// TwinCAT 3 PLC project Komplett
// ProgramVersion: 3.1.4022.1
// libraries:
//   Tc2_Standard, * (Beckhoff Automation GmbH)
//   Tc2_System, * (Beckhoff Automation GmbH)
//   Tc3_Module, * (Beckhoff Automation GmbH)
// project tree:
//   GVLs/ AN.TcGVL, DIO.TcGVL, dSub.TcGVL
//   / PlcTask.TcTTO (not stored)
//   POUs/ DoppelLauflicht.TcPOU, Komplett.TcPOU, Lauflicht.TcPOU, MAIN.TcPOU
// real-time tasks:
//   TASK PlcTask: cycle T#10ms, priority 20, ADS port 350
// motion (NC):
//   TASK NC-Task 1 SAF: cycle T#2ms, priority 4, ADS port 501
//   TASK NC-Task 1 SVB: cycle T#10ms, priority 8, ADS port 511
//   AXIS Axis 1 (id 1)
//     OtherSettings: AllowMotionCmdToSlave=true
//     encoder EncType=4
//       EncPara: MaxCount=#x0000ffff
//         Inc: RefSoftSyncMask=#x0000ffff
//     drive DrvType=24
//       Analog: ScaleFactorActTorque=0.1
//       TimeComp: TaskDelayCycles=1
//     controller CtrType=1
//       CtrPara: PriorControlFactor=1
//         Observer: BandWidth=20
//   AXIS Axis 2 (id 2)
//     OtherSettings: AllowMotionCmdToSlave=true
//     encoder EncType=4
//       EncPara: MaxCount=#x0000ffff
//         Inc: RefSoftSyncMask=#x0000ffff
//     drive DrvType=24
//       Analog: ScaleFactorActTorque=0.1
//       TimeComp: TaskDelayCycles=1
//     controller CtrType=1
//       CtrPara: PriorControlFactor=1
//         Observer: BandWidth=20
//   AXIS Axis 3 (id 3)
//     OtherSettings: AllowMotionCmdToSlave=true
//     encoder EncType=4
//       EncPara: MaxCount=#x0000ffff
//     drive DrvType=23
//       Analog: ScaleFactorActTorque=0.1
//       TimeComp: TaskDelayCycles=1
//     controller CtrType=1
//       CtrPara: PriorControlFactor=1
//         Observer: BandWidth=20
//   AXIS Axis 4 (id 4)
//     OtherSettings: AllowMotionCmdToSlave=true
//     encoder EncType=4
//       EncPara: MaxCount=#x0000ffff
//     drive DrvType=23
//       Analog: ScaleFactorActTorque=0.1
//       TimeComp: TaskDelayCycles=1
//     controller CtrType=1
//       CtrPara: PriorControlFactor=1
//         Observer: BandWidth=20
//   AXIS Axis 5 (id 5)
//     OtherSettings: AllowMotionCmdToSlave=true
//     encoder EncType=19
//       EncPara: MaxCount=#xffffffff
//     drive DrvType=16
//       DrvPara: MaxCount=#xffffffff
//         Analog: ScaleFactorActTorque=0.1
//         TimeComp: TaskDelayCycles=1
//     controller CtrType=1
//       CtrPara: PriorControlFactor=1
//         Observer: BandWidth=20
//   AXIS Axis 6 (id 6)
//     OtherSettings: AllowMotionCmdToSlave=true
//     encoder EncType=19
//       EncPara: MaxCount=#xffffffff
//     drive DrvType=16
//       DrvPara: MaxCount=#xffffffff
//         Analog: ScaleFactorActTorque=0.1
//         TimeComp: TaskDelayCycles=1
//     controller CtrType=1
//       CtrPara: PriorControlFactor=1
//         Observer: BandWidth=20
// I/O:
//   DEVICE Device 1 (EtherCAT), AmsNetId 5.35.139.20.2.1
//     Term 1 (EK1200) [EK1200-5000 EtherCAT Power supply (2A E-Bus)]
//       Term 2 (EL1809) [EL1809 16Ch. Dig. Input 24V, 3ms]
//       Term 3 (EL1809) [EL1809 16Ch. Dig. Input 24V, 3ms]
//       Term 4 (EL2809) [EL2809 16Ch. Dig. Output 24V, 0.5A]
//       Term 5 (EL2809) [EL2809 16Ch. Dig. Output 24V, 0.5A]
//       Term 6 (EL3064) [EL3064 4Ch. Ana. Input 0-10V]
//       Term 7 (EL4034) [EL4034 4Ch. Ana. Output +/-10V, 12bit]
//       Term 8 (EL7031) [EL7031 1Ch. Stepper motor output stage (24V, 1.5A)]
//       Term 9 (EL7031) [EL7031 1Ch. Stepper motor output stage (24V, 1.5A)]
//       Term 10 (EL7332) [EL7332 2Ch. DC motor output stage (24V, 1.5A)]
//       Term 11 (EL7201-0010) [EL7201-0010 1Ch. MDP742 Servo motor output stage with OCT (50V, 4A)]
//       Term 12 (EL7201-0010) [EL7201-0010 1Ch. MDP742 Servo motor output stage with OCT (50V, 4A)]
//       Term 26 (EL6090) [EL6090 Display terminal]
//       Term 27 (EK1110) [EK1110 EtherCAT extension]
// variable links:
//   NC-Task 1 SAF/Axes/Axis 1 <-> Device 1 (EtherCAT)/Term 1 (EK1200)/Term 8 (EL7031)
//     Drive/Inputs/In/nState1 @bit 3 <-> STM Status/Status/Error
//     Drive/Inputs/In/nState1 @bit 5 <-> STM Status/Status/Moving negative
//     Drive/Inputs/In/nState1 @bit 4 <-> STM Status/Status/Moving positive
//     Drive/Inputs/In/nState1 @bit 1 <-> STM Status/Status/Ready
//     Drive/Inputs/In/nState1 <-> STM Status/Status/Ready to enable
//     Drive/Inputs/In/nState1 @bit 6 <-> STM Status/Status/Torque reduced
//     Drive/Inputs/In/nState1 @bit 2 <-> STM Status/Status/Warning
//     Drive/Inputs/In/nState2 @bit 3 <-> STM Status/Status/Digital input 1
//     Drive/Inputs/In/nState2 @bit 4 <-> STM Status/Status/Digital input 2
//     Drive/Inputs/In/nState2 @bit 5 <-> STM Status/Status/Sync error
//     Drive/Inputs/In/nState2 @bit 7 <-> STM Status/Status/TxPDO Toggle
//     Drive/Inputs/In/nState4 @bit 1 <-> WcState/InputToggle
//     Drive/Inputs/In/nState4 <-> WcState/WcState
//     Drive/Outputs/Out/nCtrl1 <-> STM Control/Control/Enable
//     Drive/Outputs/Out/nCtrl1 @bit 2 <-> STM Control/Control/Reduce torque
//     Drive/Outputs/Out/nCtrl1 @bit 1 <-> STM Control/Control/Reset
//     Drive/Outputs/Out/nDataOut2[0] <-> STM Velocity/Velocity
//     Enc/Inputs/In/nDataIn1[0] <-> ENC Status compact/Counter value
//     Enc/Inputs/In/nDataIn2[0] <-> ENC Status compact/Latch value
//     Enc/Inputs/In/nState1 @bit 4 <-> ENC Status compact/Status/Counter overflow
//     Enc/Inputs/In/nState1 @bit 3 <-> ENC Status compact/Status/Counter underflow
//     Enc/Inputs/In/nState1 @bit 1 <-> ENC Status compact/Status/Latch extern valid
//     Enc/Inputs/In/nState1 @bit 2 <-> ENC Status compact/Status/Set counter done
//     Enc/Inputs/In/nState2 @bit 4 <-> ENC Status compact/Status/Status of extern latch
//     Enc/Inputs/In/nState2 @bit 5 <-> ENC Status compact/Status/Sync error
//     Enc/Inputs/In/nState2 @bit 7 <-> ENC Status compact/Status/TxPDO Toggle
//     Enc/Inputs/In/nState4 @bit 1 <-> WcState/InputToggle
//     Enc/Inputs/In/nState4 <-> WcState/WcState
//     Enc/Outputs/Out/nCtrl1 @bit 3 <-> ENC Control compact/Control/Enable latch extern on negative edge
//     Enc/Outputs/Out/nCtrl1 @bit 1 <-> ENC Control compact/Control/Enable latch extern on positive edge
//     Enc/Outputs/Out/nCtrl1 @bit 2 <-> ENC Control compact/Control/Set counter
//     Enc/Outputs/Out/nDataOut1[0] <-> ENC Control compact/Set counter value
//   NC-Task 1 SAF/Axes/Axis 2 <-> Device 1 (EtherCAT)/Term 1 (EK1200)/Term 9 (EL7031)
//     Drive/Inputs/In/nState1 @bit 3 <-> STM Status/Status/Error
//     Drive/Inputs/In/nState1 @bit 5 <-> STM Status/Status/Moving negative
//     Drive/Inputs/In/nState1 @bit 4 <-> STM Status/Status/Moving positive
//     Drive/Inputs/In/nState1 @bit 1 <-> STM Status/Status/Ready
//     Drive/Inputs/In/nState1 <-> STM Status/Status/Ready to enable
//     Drive/Inputs/In/nState1 @bit 6 <-> STM Status/Status/Torque reduced
//     Drive/Inputs/In/nState1 @bit 2 <-> STM Status/Status/Warning
//     Drive/Inputs/In/nState2 @bit 3 <-> STM Status/Status/Digital input 1
//     Drive/Inputs/In/nState2 @bit 4 <-> STM Status/Status/Digital input 2
//     Drive/Inputs/In/nState2 @bit 5 <-> STM Status/Status/Sync error
//     Drive/Inputs/In/nState2 @bit 7 <-> STM Status/Status/TxPDO Toggle
//     Drive/Inputs/In/nState4 @bit 1 <-> WcState/InputToggle
//     Drive/Inputs/In/nState4 <-> WcState/WcState
//     Drive/Outputs/Out/nCtrl1 <-> STM Control/Control/Enable
//     Drive/Outputs/Out/nCtrl1 @bit 2 <-> STM Control/Control/Reduce torque
//     Drive/Outputs/Out/nCtrl1 @bit 1 <-> STM Control/Control/Reset
//     Drive/Outputs/Out/nDataOut2[0] <-> STM Velocity/Velocity
//     Enc/Inputs/In/nDataIn1[0] <-> ENC Status compact/Counter value
//     Enc/Inputs/In/nDataIn2[0] <-> ENC Status compact/Latch value
//     Enc/Inputs/In/nState1 @bit 4 <-> ENC Status compact/Status/Counter overflow
//     Enc/Inputs/In/nState1 @bit 3 <-> ENC Status compact/Status/Counter underflow
//     Enc/Inputs/In/nState1 @bit 1 <-> ENC Status compact/Status/Latch extern valid
//     Enc/Inputs/In/nState1 @bit 2 <-> ENC Status compact/Status/Set counter done
//     Enc/Inputs/In/nState2 @bit 4 <-> ENC Status compact/Status/Status of extern latch
//     Enc/Inputs/In/nState2 @bit 5 <-> ENC Status compact/Status/Sync error
//     Enc/Inputs/In/nState2 @bit 7 <-> ENC Status compact/Status/TxPDO Toggle
//     Enc/Inputs/In/nState4 @bit 1 <-> WcState/InputToggle
//     Enc/Inputs/In/nState4 <-> WcState/WcState
//     Enc/Outputs/Out/nCtrl1 @bit 3 <-> ENC Control compact/Control/Enable latch extern on negative edge
//     Enc/Outputs/Out/nCtrl1 @bit 1 <-> ENC Control compact/Control/Enable latch extern on positive edge
//     Enc/Outputs/Out/nCtrl1 @bit 2 <-> ENC Control compact/Control/Set counter
//     Enc/Outputs/Out/nDataOut1[0] <-> ENC Control compact/Set counter value
//   NC-Task 1 SAF/Axes/Axis 3 <-> Device 1 (EtherCAT)/Term 1 (EK1200)/Term 10 (EL7332)
//     Drive/Inputs/In/nState1 @bit 3 <-> DCM Status Channel 1/Status/Error
//     Drive/Inputs/In/nState1 @bit 5 <-> DCM Status Channel 1/Status/Moving negative
//     Drive/Inputs/In/nState1 @bit 4 <-> DCM Status Channel 1/Status/Moving positive
//     Drive/Inputs/In/nState1 @bit 1 <-> DCM Status Channel 1/Status/Ready
//     Drive/Inputs/In/nState1 <-> DCM Status Channel 1/Status/Ready to enable
//     Drive/Inputs/In/nState1 @bit 6 <-> DCM Status Channel 1/Status/Torque reduced
//     Drive/Inputs/In/nState1 @bit 2 <-> DCM Status Channel 1/Status/Warning
//     Drive/Inputs/In/nState2 @bit 3 <-> DCM Status Channel 1/Status/Digital input 1
//     Drive/Inputs/In/nState2 @bit 4 <-> DCM Status Channel 1/Status/Digital input 2
//     Drive/Inputs/In/nState2 @bit 5 <-> DCM Status Channel 1/Status/Sync error
//     Drive/Inputs/In/nState2 @bit 7 <-> DCM Status Channel 1/Status/TxPDO Toggle
//     Drive/Inputs/In/nState4 @bit 1 <-> WcState/InputToggle
//     Drive/Inputs/In/nState4 <-> WcState/WcState
//     Drive/Outputs/Out/nCtrl1 <-> DCM Control Channel 1/Control/Enable
//     Drive/Outputs/Out/nCtrl1 @bit 2 <-> DCM Control Channel 1/Control/Reduce torque
//     Drive/Outputs/Out/nCtrl1 @bit 1 <-> DCM Control Channel 1/Control/Reset
//     Drive/Outputs/Out/nDataOut2[0] <-> DCM Velocity Channel 1/Velocity
//   NC-Task 1 SAF/Axes/Axis 4 <-> Device 1 (EtherCAT)/Term 1 (EK1200)/Term 10 (EL7332)
//     Drive/Inputs/In/nState1 @bit 3 <-> DCM Status Channel 2/Status/Error
//     Drive/Inputs/In/nState1 @bit 5 <-> DCM Status Channel 2/Status/Moving negative
//     Drive/Inputs/In/nState1 @bit 4 <-> DCM Status Channel 2/Status/Moving positive
//     Drive/Inputs/In/nState1 @bit 1 <-> DCM Status Channel 2/Status/Ready
//     Drive/Inputs/In/nState1 <-> DCM Status Channel 2/Status/Ready to enable
//     Drive/Inputs/In/nState1 @bit 6 <-> DCM Status Channel 2/Status/Torque reduced
//     Drive/Inputs/In/nState1 @bit 2 <-> DCM Status Channel 2/Status/Warning
//     Drive/Inputs/In/nState2 @bit 3 <-> DCM Status Channel 2/Status/Digital input 1
//     Drive/Inputs/In/nState2 @bit 4 <-> DCM Status Channel 2/Status/Digital input 2
//     Drive/Inputs/In/nState2 @bit 5 <-> DCM Status Channel 2/Status/Sync error
//     Drive/Inputs/In/nState2 @bit 7 <-> DCM Status Channel 2/Status/TxPDO Toggle
//     Drive/Inputs/In/nState4 @bit 1 <-> WcState/InputToggle
//     Drive/Inputs/In/nState4 <-> WcState/WcState
//     Drive/Outputs/Out/nCtrl1 <-> DCM Control Channel 2/Control/Enable
//     Drive/Outputs/Out/nCtrl1 @bit 2 <-> DCM Control Channel 2/Control/Reduce torque
//     Drive/Outputs/Out/nCtrl1 @bit 1 <-> DCM Control Channel 2/Control/Reset
//     Drive/Outputs/Out/nDataOut2[0] <-> DCM Velocity Channel 2/Velocity
//   NC-Task 1 SAF/Axes/Axis 5 <-> Device 1 (EtherCAT)/Term 1 (EK1200)/Term 11 (EL7201-0010)
//     Drive/Inputs/In/nDcOutputTime <-> InfoData/DcOutputShift
//     Drive/Inputs/In/nState1 <-> DRV Statusword/Statusword
//     Drive/Inputs/In/nState2 <-> DRV Statusword/Statusword @bit 8
//     Drive/Inputs/In/nState4 @bit 1 <-> WcState/InputToggle
//     Drive/Inputs/In/nState4 <-> WcState/WcState
//     Drive/Outputs/Out/nCtrl1 <-> DRV Controlword/Controlword
//     Drive/Outputs/Out/nCtrl2 <-> DRV Controlword/Controlword @bit 8
//     Drive/Outputs/Out/nDataOut2 <-> DRV Target velocity/Target velocity
//     Enc/Inputs/In/nDataIn1 <-> FB Position/Position
//     Enc/Inputs/In/nDcInputTime <-> InfoData/DcInputShift
//     Enc/Inputs/In/nState4 @bit 1 <-> WcState/InputToggle
//     Enc/Inputs/In/nState4 <-> WcState/WcState
//   NC-Task 1 SAF/Axes/Axis 6 <-> Device 1 (EtherCAT)/Term 1 (EK1200)/Term 12 (EL7201-0010)
//     Drive/Inputs/In/nDcOutputTime <-> InfoData/DcOutputShift
//     Drive/Inputs/In/nState1 <-> DRV Statusword/Statusword
//     Drive/Inputs/In/nState2 <-> DRV Statusword/Statusword @bit 8
//     Drive/Inputs/In/nState4 @bit 1 <-> WcState/InputToggle
//     Drive/Inputs/In/nState4 <-> WcState/WcState
//     Drive/Outputs/Out/nCtrl1 <-> DRV Controlword/Controlword
//     Drive/Outputs/Out/nCtrl2 <-> DRV Controlword/Controlword @bit 8
//     Drive/Outputs/Out/nDataOut2 <-> DRV Target velocity/Target velocity
//     Enc/Inputs/In/nDataIn1 <-> FB Position/Position
//     Enc/Inputs/In/nDcInputTime <-> InfoData/DcInputShift
//     Enc/Inputs/In/nState4 @bit 1 <-> WcState/InputToggle
//     Enc/Inputs/In/nState4 <-> WcState/WcState
//   Komplett/Komplett Instance <-> Device 1 (EtherCAT)/Term 1 (EK1200)/Term 2 (EL1809)
//     PlcTask Inputs/dSub.B1 <-> Channel 1/Input
//     PlcTask Inputs/dSub.B2 <-> Channel 2/Input
//     PlcTask Inputs/dSub.S1 <-> Channel 4/Input
//     PlcTask Inputs/dSub.S10 <-> Channel 12/Input
//     PlcTask Inputs/dSub.S11 <-> Channel 13/Input
//     PlcTask Inputs/dSub.S12 <-> Channel 14/Input
//     PlcTask Inputs/dSub.S13 <-> Channel 15/Input
//     PlcTask Inputs/dSub.S14 <-> Channel 16/Input
//     PlcTask Inputs/dSub.S2 <-> Channel 3/Input
//     PlcTask Inputs/dSub.S3 <-> Channel 6/Input
//     PlcTask Inputs/dSub.S4 <-> Channel 5/Input
//     PlcTask Inputs/dSub.S5 <-> Channel 8/Input
//     PlcTask Inputs/dSub.S6 <-> Channel 7/Input
//     PlcTask Inputs/dSub.S7 <-> Channel 10/Input
//     PlcTask Inputs/dSub.S8 <-> Channel 9/Input
//     PlcTask Inputs/dSub.S9 <-> Channel 11/Input
//   Komplett/Komplett Instance <-> Device 1 (EtherCAT)/Term 1 (EK1200)/Term 3 (EL1809)
//     PlcTask Inputs/DIO.DI_{1..16} <-> Channel {1..16}/Input  (16 links)
//   Komplett/Komplett Instance <-> Device 1 (EtherCAT)/Term 1 (EK1200)/Term 4 (EL2809)
//     PlcTask Outputs/dSub.P{1..14} <-> Channel {3..16}/Output  (14 links)
//     PlcTask Outputs/dSub.Q1 <-> Channel 1/Output
//     PlcTask Outputs/dSub.Q2 <-> Channel 2/Output
//   Komplett/Komplett Instance <-> Device 1 (EtherCAT)/Term 1 (EK1200)/Term 5 (EL2809)
//     PlcTask Outputs/DIO.DQ_{1..16} <-> Channel {1..16}/Output  (16 links)
//   Komplett/Komplett Instance <-> Device 1 (EtherCAT)/Term 1 (EK1200)/Term 6 (EL3064)
//     PlcTask Inputs/AN.AI_1 <-> AI Standard Channel 3/Value
//     PlcTask Inputs/AN.AI_2 <-> AI Standard Channel 4/Value
//     PlcTask Inputs/dSub.AI_0 <-> AI Standard Channel 1/Value
//     PlcTask Inputs/dSub.AI_1 <-> AI Standard Channel 2/Value
//   Komplett/Komplett Instance <-> Device 1 (EtherCAT)/Term 1 (EK1200)/Term 7 (EL4034)
//     PlcTask Outputs/AN.AQ_1 <-> AO Outputs Channel 3/Analog output
//     PlcTask Outputs/AN.AQ_2 <-> AO Outputs Channel 4/Analog output
//     PlcTask Outputs/dSub.AQ_0 <-> AO Outputs Channel 1/Analog output

// ---- GVLs/AN.TcGVL
{attribute 'qualified_only'}
VAR_GLOBAL	
	AI_1 AT %I*: INT;	// Analogeingang AI 1	
 	AI_2 AT %I*: INT;	// Analogeingang AI 2		
	AQ_1 AT %Q*: INT;	// Analogausgang AQ 1	 
	AQ_2 AT %Q*: INT;	// Analogausgang AQ 2	
END_VAR

// ---- GVLs/DIO.TcGVL
{attribute 'qualified_only'}
VAR_GLOBAL
	
	DI_1 AT %IX1620.0: BOOL; 	// Digitaler Eingang 1	
	DI_2 AT %IX1620.1: BOOL; 	// Digitaler Eingang 2	
	DI_3 AT %IX1620.2: BOOL; 	// Digitaler Eingang 3	
	DI_4 AT %IX1620.3: BOOL; 	// Digitaler Eingang 4		
	DI_5 AT %IX1620.4: BOOL; 	// Digitaler Eingang 5	
	DI_6 AT %IX1620.5: BOOL; 	// Digitaler Eingang 6	
	DI_7 AT %IX1620.6: BOOL; 	// Digitaler Eingang 7	
	DI_8 AT %IX1620.7: BOOL; 	// Digitaler Eingang 8	
	DI_9 AT %IX1621.0: BOOL; 	// Digitaler Eingang 9	
	DI_10 AT %IX1621.1: BOOL; 	// Digitaler Eingang 10		
	DI_11 AT %IX1621.2: BOOL; 	// Digitaler Eingang 11	
	DI_12 AT %IX1621.3: BOOL; 	// Digitaler Eingang 12			
	DI_13 AT %IX1621.4: BOOL; 	// Digitaler Eingang 13	
	DI_14 AT %IX1621.5: BOOL; 	// Digitaler Eingang 14	
	DI_15 AT %IX1621.6: BOOL; 	// Digitaler Eingang 15	
	DI_16 AT %IX1621.7: BOOL; 	// Digitaler Eingang 16	
	
	DQ_1 AT %QX1588.0: BOOL; 	// Digitaler Ausgang 1	
	DQ_2 AT %QX1588.1: BOOL; 	// Digitaler Ausgang 2	
	DQ_3 AT %QX1588.2: BOOL; 	// Digitaler Ausgang 3	
	DQ_4 AT %QX1588.3: BOOL; 	// Digitaler Ausgang 4	
	DQ_5 AT %QX1588.4: BOOL; 	// Digitaler Ausgang 5	
	DQ_6 AT %QX1588.5: BOOL; 	// Digitaler Ausgang 6	
	DQ_7 AT %QX1588.6: BOOL; 	// Digitaler Ausgang 7	
	DQ_8 AT %QX1588.7: BOOL; 	// Digitaler Ausgang 8	
	DQ_9 AT %QX1589.0: BOOL; 	// Digitaler Ausgang 9	
	DQ_10 AT %QX1589.1: BOOL; 	// Digitaler Ausgang 10	
	DQ_11 AT %QX1589.2: BOOL; 	// Digitaler Ausgang 11	
	DQ_12 AT %QX1589.3: BOOL; 	// Digitaler Ausgang 12		
	DQ_13 AT %QX1589.4: BOOL; 	// Digitaler Ausgang 13	
	DQ_14 AT %QX1589.5: BOOL; 	// Digitaler Ausgang 14	 	
	DQ_15 AT %QX1589.6: BOOL; 	// Digitaler Ausgang 15	
	DQ_16 AT %QX1589.7: BOOL; 	// Digitaler Ausgang 16	

	DIB_1_8 AT %IB1620: BYTE;	// Digitale Eingänge 1..8
	DIB_9_16 AT %IB1621: BYTE;	// Digitale Eingänge 9..16	
	DIW_1_16 AT %IB1620: WORD;	// Digitale Eingänge 1..16
	
	DQB_1_8 AT %QB1588: BYTE;	// Digitale Ausgänge 1..8
	DQB_9_16 AT %QB1589: BYTE;	// Digitale Ausgänge 9..16
	DQW_1_16 AT %QB1588: WORD;	// Digitale Ausgänge 1..16
END_VAR

// ---- GVLs/dSub.TcGVL
{attribute 'qualified_only'}
VAR_GLOBAL	
	// ACHTUNG für die Linearachse sind die Ein- und Ausgänge richtig eingetragen!
	B1 AT %IX1618.0: BOOL; 		// Linearantrieb Endlage links (Öffner)
	B2 AT %IX1618.1: BOOL;		// Linearantrieb Endlage rechts (Öffner)
	S2 AT %IX1618.2: BOOL;		// Taster (0) (Öffner)
	S1 AT %IX1618.3: BOOL;		// Taster (1) (Schliesser)
	S4 AT %IX1618.4: BOOL;		// Taster II (Schliesser)
	S3 AT %IX1618.5: BOOL;		// Taster I (Schliesser)
	S6 AT %IX1618.6: BOOL;		// Taster Pfeil ab (Schliesser)
	S5 AT %IX1618.7: BOOL;		// Taster Pfeil auf (Schliesser)
	S8 AT %IX1619.0: BOOL;		// Taster - (Schliesser)
	S7 AT %IX1619.1: BOOL;		// Taster + (Schliesser)
	S9 AT %IX1619.2: BOOL;		// Taster STOP (Öffner)	
	S10 AT %IX1619.3: BOOL;		// Taster Not Halt (Öffner)	
	S11 AT %IX1619.4: BOOL;		// Taster Not Halt (Schliesser)
	S12 AT %IX1619.5: BOOL;		//
	S13 AT %IX1619.6: BOOL;		//
	S14 AT %IX1619.7: BOOL;		//
	
	Q1 AT %QX1586.0: BOOL;		// Linearantrieb Rechtslauf
	Q2 AT %QX1586.1: BOOL;		// Linearantrieb Linkslauf
	P1 AT %QX1586.2: BOOL;		// Meldeleuchte im Taster S1 (weiß)
	P2 AT %QX1586.3: BOOL;		// Meldeleuchte weiß
	P3 AT %QX1586.4: BOOL;		// Meldeleuchte rot
	P4 AT %QX1586.5: BOOL;		// Meldeleuchte grün	
	P5 AT %QX1586.6: BOOL;		//
	P6 AT %QX1586.7: BOOL;		//
	P7 AT %QX1587.0: BOOL;		//
	P8 AT %QX1587.1: BOOL;		//
	P9 AT %QX1587.2: BOOL;		//
	P10 AT %QX1587.3: BOOL;		//
	P11 AT %QX1587.4: BOOL;		//
	P12 AT %QX1587.5: BOOL;		//
	P13 AT %QX1587.6: BOOL;		//
	P14 AT %QX1587.7: BOOL;		//
	
	DIB_1_8 AT %IB1618: BYTE;	// Digitale Eingänge 1..8
	DIB_9_16 AT %IB1619: BYTE;	// Digitale Eingänge 9..16
	
	DIW_1_16 AT %IB1618: WORD;	// Digitale Eingänge 1..16
	
	DQB_1_8 AT %QB1586: BYTE;	// Digitale Ausgänge 1..8
	DQB_9_16 AT %QB1587: BYTE;	// Digitale Ausgänge 9..16

	DQW_1_16 AT %QB1586: WORD;	// Digitale Ausgänge 1..16	
		
	AI_0 AT %I*: INT;			// Analogeingang 0
	AI_1 AT %I*: INT;			// Analogeingang 1
	
	AQ_0 AT %Q*: INT;			// Analogausgang 0	
END_VAR

// ---- POUs/DoppelLauflicht.TcPOU
FUNCTION_BLOCK DoppelLauflicht
VAR_INPUT
END_VAR
VAR_OUTPUT
END_VAR
VAR
	Blinker: TON;
	Zaehler : WORD;
END_VAR


Blinker(IN:= NOT Blinker.Q, PT:= T#100MS );

IF Blinker.Q THEN	Zaehler := Zaehler + 1;END_IF
IF Zaehler > 7 THEN Zaehler := 0;END_IF

dSub.DQB_1_8 := SHL(1, Zaehler);
dSub.DQB_9_16 := SHL(1, 7 - Zaehler);

END_FUNCTION_BLOCK

// ---- POUs/Komplett.TcPOU
FUNCTION_BLOCK Komplett
VAR_INPUT
END_VAR
VAR_OUTPUT
END_VAR
VAR
	Timer1: TON;
END_VAR

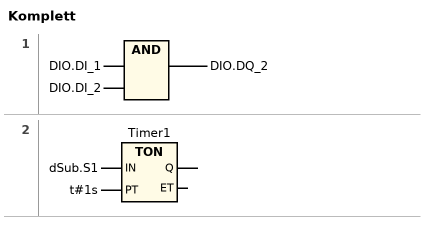
// NETWORK 1
DIO.DQ_2 := DIO.DI_1 AND DIO.DI_2;

// NETWORK 2
Timer1(IN := dSub.S1, PT := t#1s); // TON

END_FUNCTION_BLOCK

// ---- POUs/Lauflicht.TcPOU
FUNCTION_BLOCK Lauflicht
VAR_INPUT
END_VAR
VAR_OUTPUT
END_VAR
VAR
	Blinker: TON;
	Zaehler : WORD;
END_VAR

Blinker(IN:= NOT Blinker.Q, PT:= T#100MS );

IF Blinker.Q THEN	Zaehler := Zaehler + 1;END_IF
IF Zaehler > 15 THEN Zaehler := 0;END_IF

DIO.DQW_1_16 := SHL(1 ,Zaehler);

END_FUNCTION_BLOCK

// ---- POUs/MAIN.TcPOU
PROGRAM MAIN
VAR
	Komplett: Komplett;
	Lauflicht:Lauflicht;
	DoppelLauflicht: DoppelLauflicht;
END_VAR


Komplett();
Lauflicht();
DoppelLauflicht();

END_PROGRAM
